# EPICS substitutions: apps/plcApp/Db/cryodbox_torus_comm.substitutions
#
# cryodbox_torus_comm.substitutions
#
# Author: Wesley Moore (wmoore@jlab.org)
# Date:   June 2017
#

file "db/torus_bi_generic.db" { pattern
    { PLCID,    P,        R,    TAG,            ZNAM,  ONAM,    ZSV,        OSV,        DESC }
    { PLC_CRYO, B_TORUS:, DBX:, UPS_On_Battery, Ok,    Warning, NO_ALARM,   MAJOR,      "PLC On UPS Battery" }
    { PLC_CRYO, B_TORUS:, DBX:, FAULT_24VDC,    Fault, Ok,      MAJOR,      NO_ALARM,   "Rhino 24VDC PSU Status" }
}
